PROGRAM oArmSlowPullHomingCtrl
VAR

	ArmSlowPullHomingFB: fbMotorHomingAxis;
	ArmSlowPullHomeWord: CMP_OC_DW;

	bSlowPullResetBit: BOOL;

	LifterReadStatus: MC_ReadStatus;
	LifterReset: MC_Reset;
	LifterSoeReset: FB_SoEReset;

END_VAR

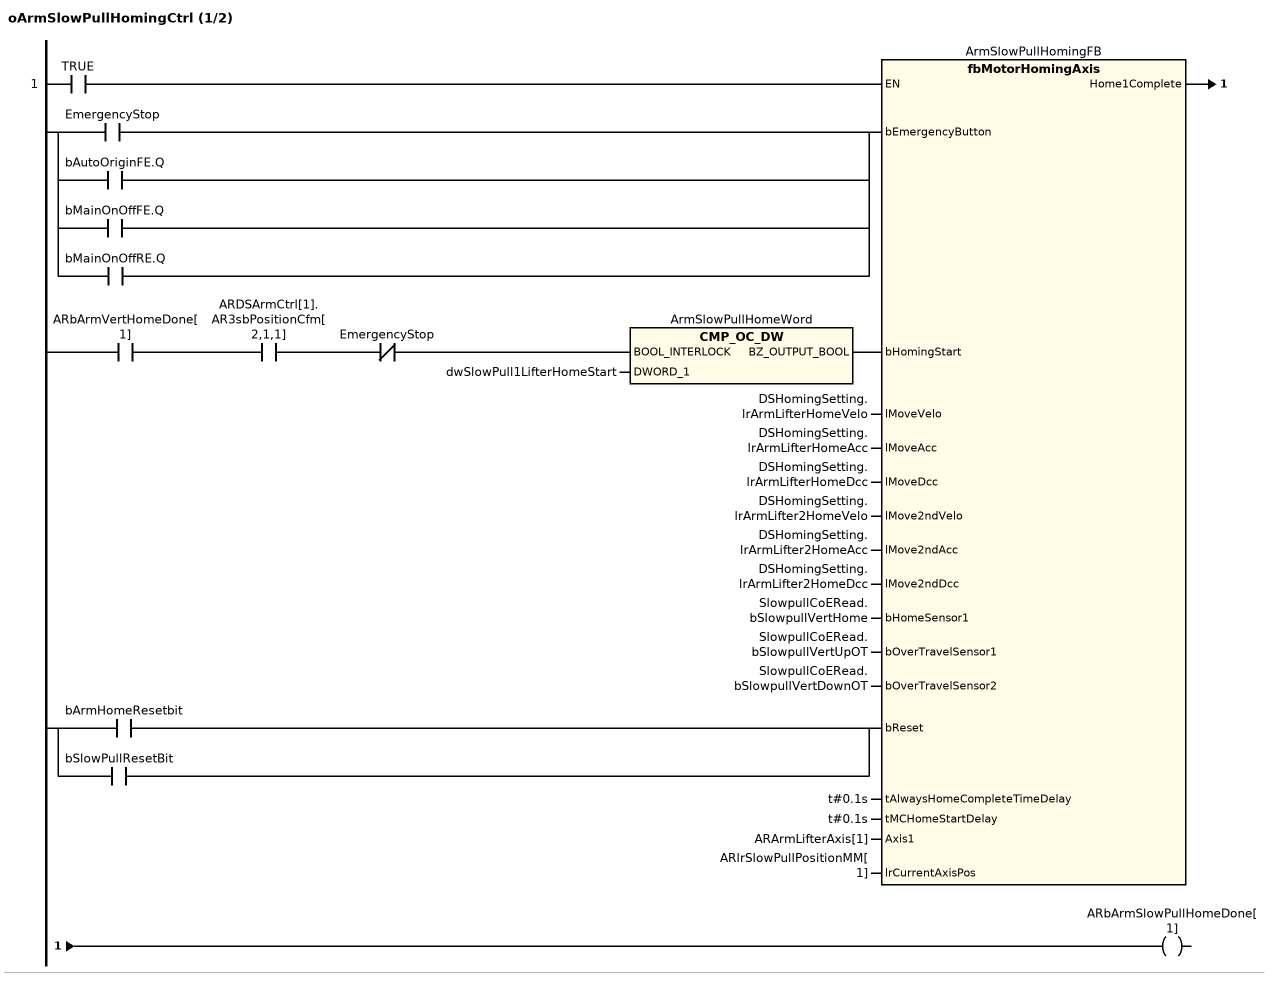
// NETWORK 1
ArmSlowPullHomeWord(BOOL_INTERLOCK := ARbArmVertHomeDone[1] AND ARDSArmCtrl[1].AR3sbPositionCfm[2,1,1] AND NOT EmergencyStop, DWORD_1 := dwSlowPull1LifterHomeStart); // CMP_OC_DW
ArmSlowPullHomingFB(
    bEmergencyButton := EmergencyStop OR bAutoOriginFE.Q OR bMainOnOffFE.Q OR bMainOnOffRE.Q,
    bHomingStart := ArmSlowPullHomeWord.BZ_OUTPUT_BOOL,
    lMoveVelo := DSHomingSetting.lrArmLifterHomeVelo,
    lMoveAcc := DSHomingSetting.lrArmLifterHomeAcc,
    lMoveDcc := DSHomingSetting.lrArmLifterHomeDcc,
    lMove2ndVelo := DSHomingSetting.lrArmLifter2HomeVelo,
    lMove2ndAcc := DSHomingSetting.lrArmLifter2HomeAcc,
    lMove2ndDcc := DSHomingSetting.lrArmLifter2HomeDcc,
    bHomeSensor1 := SlowpullCoERead.bSlowpullVertHome,
    bOverTravelSensor1 := SlowpullCoERead.bSlowpullVertUpOT,
    bOverTravelSensor2 := SlowpullCoERead.bSlowpullVertDownOT,
    bReset := bArmHomeResetbit OR bSlowPullResetBit,
    tAlwaysHomeCompleteTimeDelay := t#0.1s,
    tMCHomeStartDelay := t#0.1s,
    Axis1 := ARArmLifterAxis[1],
    lrCurrentAxisPos := ARlrSlowPullPositionMM[1]); // fbMotorHomingAxis
ARbArmSlowPullHomeDone[1] := ArmSlowPullHomingFB.Home1Complete;

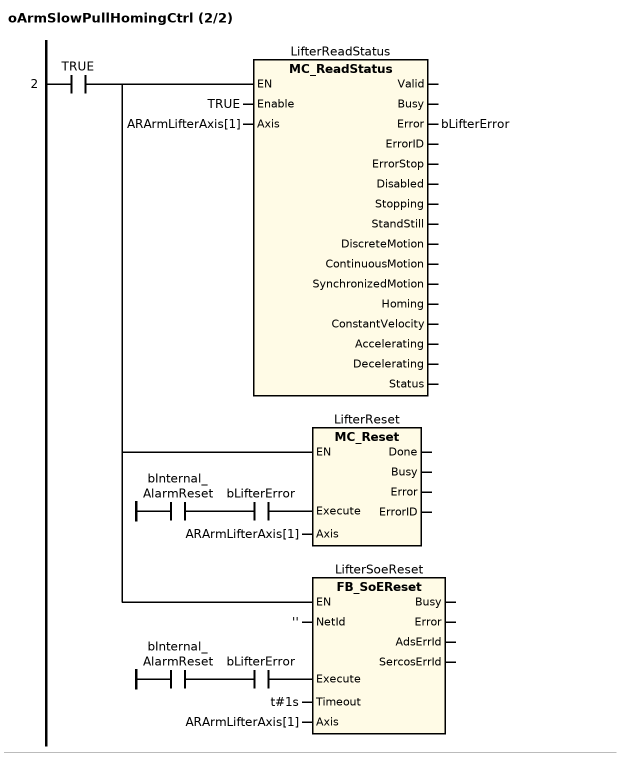
// NETWORK 2
LifterReadStatus(Enable := TRUE, Axis := ARArmLifterAxis[1], Error => bLifterError); // MC_ReadStatus
LifterReset(Execute := bInternal_AlarmReset AND bLifterError, Axis := ARArmLifterAxis[1]); // MC_Reset
LifterSoeReset(
    NetId := '',
    Execute := bInternal_AlarmReset AND bLifterError,
    Timeout := t#1s,
    Axis := ARArmLifterAxis[1]); // FB_SoEReset

END_PROGRAM

(* stored: Version 1.1.0.1, ProductVersion 3.1.4024.12
   POU oArmSlowPullHomingCtrl: Id {3f49be05-6b0a-478e-9c71-de0855efc3a5}, SpecialFunc None *)
